// Mitsubishi GX Works2 project: Project1   PLC: FX3G

// global labels: Global1
VAR_GLOBAL
  StartWorkDay AT X007 : BOOL;
  TurnLightAssist AT X011 : BOOL;
  CurrentlyWorking AT Y007 : BOOL;
  yeastInput AT D1100 : REAL;
  yeastInventory AT D1108 : REAL;
  maltInput AT D1102 : REAL;
  maltInventory AT D1110 : REAL;
  hopsInput AT D1104 : REAL;
  hopsInventory AT D1112 : REAL;
  readyBeerPacks AT D1106 : INT;
  startCookingPhase AT X001 : BOOL;
END_VAR
VAR_GLOBAL CONSTANT
  pilsnerMin : INT := 6;
END_VAR
VAR_GLOBAL
  analogInput AT D8280 : INT;
END_VAR
VAR_GLOBAL CONSTANT
  cont400 : INT := 400;
END_VAR
VAR_GLOBAL
  saveAnalog AT D7000 : INT;
  pilsnerCheckAssist AT M0 : BOOL;
  lagerCheckAssist AT M1 : BOOL;
END_VAR
VAR_GLOBAL CONSTANT
  yeastPilsnerMin : REAL := 120;
  maltPilsnerMin : REAL := 6;
  hopsPilsnerMin : REAL := 53;
  cookingTime : INT := 400;
END_VAR
VAR_GLOBAL
  yesPilsnerInventory AT M16 : BOOL;
  CookingTimer AT TC1 : BOOL;
END_VAR
VAR_GLOBAL CONSTANT
  DoneCooking : INT := 40;
END_VAR
VAR_GLOBAL
  Cooking AT TS1 : BOOL;
  CookingProcess AT Y001 : BOOL;
END_VAR
VAR_GLOBAL CONSTANT
  yeastLagerMin : REAL := 150;
  maltLagerMin : REAL := 12;
  hopsLagerMin : REAL := 60;
END_VAR
VAR_GLOBAL
  yesLagerInventory AT M17 : BOOL;
END_VAR
VAR_GLOBAL CONSTANT
  lagerMax : INT := 5;
END_VAR
VAR_GLOBAL
  startFermPhase AT X005 : BOOL;
END_VAR
VAR_GLOBAL CONSTANT
  doneFermPilsner : INT := 40;
END_VAR
VAR_GLOBAL
  FermPilsner AT TC3 : BOOL;
  FermLager AT TC5 : BOOL;
END_VAR
VAR_GLOBAL CONSTANT
  doneFermLager : INT := 30;
END_VAR
VAR_GLOBAL
  FermPilsnerDone AT TS3 : BOOL;
  FermLagerDone AT TS5 : BOOL;
  startBlinking AT M20 : BOOL;
  blinkingHelp AT M21 : BOOL;
  blinkY3 AT TC2 : BOOL;
END_VAR
VAR_GLOBAL CONSTANT
  blinkTime : INT := 5;
END_VAR
VAR_GLOBAL
  blink1 AT TS2 : BOOL;
  lightY3 AT Y003 : BOOL;
  blinkY4 AT TC4 : BOOL;
  blink2 AT TS4 : BOOL;
  lightY4 AT Y004 : BOOL;
  startPackPhase AT X002 : BOOL;
  packBottle AT X000 : BOOL;
  bottlesNum AT CC1 : BOOL;
END_VAR
VAR_GLOBAL CONSTANT
  bottlesPacked : INT := 1;
END_VAR
VAR_GLOBAL
  sixPackNum AT CC2 : BOOL;
END_VAR
VAR_GLOBAL CONSTANT
  sixPacksPacked : INT := 6;
END_VAR
VAR_GLOBAL
  oneBottlePacked AT CS1 : BOOL;
  duringPacking AT Y002 : BOOL;
  doneSixPack AT CS2 : BOOL;
END_VAR
VAR_GLOBAL CONSTANT
  addSixPack : INT := 1;
END_VAR
VAR_GLOBAL
  lackOfProducts AT M19 : BOOL;
  doneSixPacks AT CS2 : BOOL;
  checkYeastForPilsner AT M22 : BOOL;
  checkMaltForPilsner AT M23 : BOOL;
  checkHopsForPilsner AT M24 : BOOL;
  checkYeastForLager AT M25 : BOOL;
  checkMaltForLager AT M26 : BOOL;
  checkHopsForLager AT M27 : BOOL;
  checkYeastForPilsnerEnd AT M70 : BOOL;
  checkMaltForPilsnerEnd AT M71 : BOOL;
  checkHopsForPilsnerEnd AT M72 : BOOL;
  checkYeastForLagerEnd AT M73 : BOOL;
  checkMaltForLagerEnd AT M74 : BOOL;
  checkHopsForLagerEnd AT M75 : BOOL;
  startAnalogOutput AT M100 : BOOL;
END_VAR
VAR_GLOBAL CONSTANT
  constDivide : INT := 40;
END_VAR
VAR_GLOBAL
  analogOutput AT D8282 : INT;
  lackOfProductsEnd AT M50 : BOOL;
END_VAR

// task Task_01 (event TRUE, interval 0, priority 31): POU_01

PROGRAM POU_01
(* structured ladder/FBD written out as ST: instructions are called as NAME(EN, inputs, outputs); _pN, _eN, _tN stand for wires *)
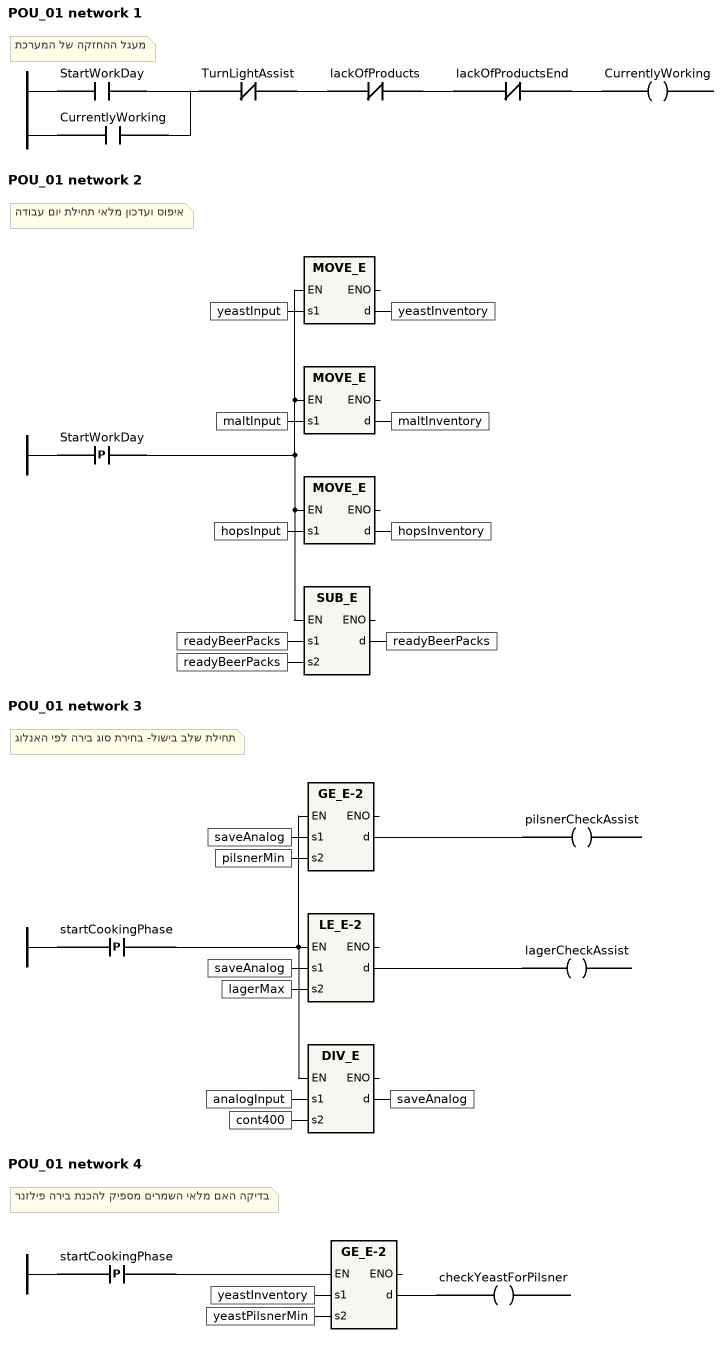
(* network 1 *)
(* מעגל ההחזקה של המערכת *)
CurrentlyWorking := (((StartWorkDay OR CurrentlyWorking) AND NOT TurnLightAssist) AND NOT lackOfProducts) AND NOT lackOfProductsEnd;
(* network 2 *)
(* איפוס ועדכון מלאי תחילת יום עבודה *)
_p1 := LDP(TRUE, StartWorkDay);
MOVE_E(_p1, yeastInput, yeastInventory);
MOVE_E(_p1, maltInput, maltInventory);
MOVE_E(_p1, hopsInput, hopsInventory);
SUB_E(_p1, readyBeerPacks, readyBeerPacks, readyBeerPacks);
(* network 3 *)
(* תחילת שלב בישול- בחירת סוג בירה לפי האנלוג *)
_p1 := LDP(TRUE, startCookingPhase);
DIV_E(_p1, analogInput, cont400, saveAnalog);
GE_E(_p1, saveAnalog, pilsnerMin, _t2);
pilsnerCheckAssist := _t2;
LE_E(_p1, saveAnalog, lagerMax, _t3);
lagerCheckAssist := _t3;
(* network 4 *)
(* בדיקה האם מלאי השמרים מספיק להכנת בירה פילזנר *)
GE_E(LDP(TRUE, startCookingPhase), yeastInventory, yeastPilsnerMin, _t1);
checkYeastForPilsner := _t1;
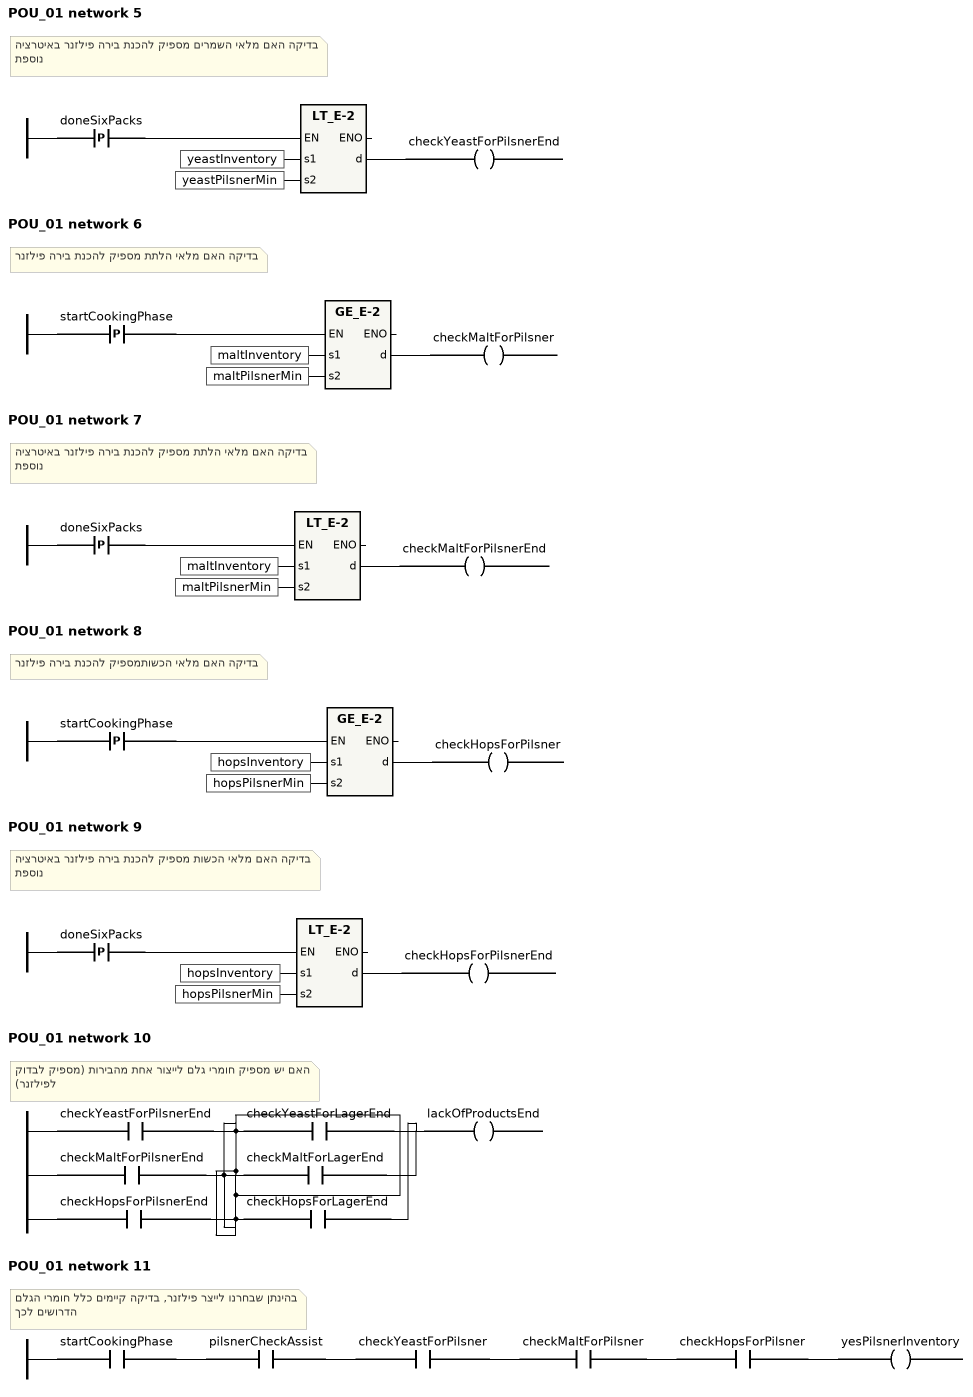
(* network 5 *)
(* בדיקה האם מלאי השמרים מספיק להכנת בירה פילזנר באיטרציה נוספת *)
LT_E(LDP(TRUE, doneSixPacks), yeastInventory, yeastPilsnerMin, _t1);
checkYeastForPilsnerEnd := _t1;
(* network 6 *)
(* בדיקה האם מלאי הלתת מספיק להכנת בירה פילזנר *)
GE_E(LDP(TRUE, startCookingPhase), maltInventory, maltPilsnerMin, _t1);
checkMaltForPilsner := _t1;
(* network 7 *)
(* בדיקה האם מלאי הלתת מספיק להכנת בירה פילזנר באיטרציה נוספת *)
LT_E(LDP(TRUE, doneSixPacks), maltInventory, maltPilsnerMin, _t1);
checkMaltForPilsnerEnd := _t1;
(* network 8 *)
(* בדיקה האם מלאי הכשותמספיק להכנת בירה פילזנר *)
GE_E(LDP(TRUE, startCookingPhase), hopsInventory, hopsPilsnerMin, _t1);
checkHopsForPilsner := _t1;
(* network 9 *)
(* בדיקה האם מלאי הכשות מספיק להכנת בירה פילזנר באיטרציה נוספת *)
LT_E(LDP(TRUE, doneSixPacks), hopsInventory, hopsPilsnerMin, _t1);
checkHopsForPilsnerEnd := _t1;
(* network 10 *)
(* האם יש מספיק חומרי גלם לייצור אחת מהבירות (מספיק לבדוק לפילזנר) *)
_p1 := checkYeastForPilsnerEnd OR checkMaltForPilsnerEnd OR checkHopsForPilsnerEnd;
lackOfProductsEnd := (_p1 AND checkYeastForLagerEnd) OR (_p1 AND checkMaltForLagerEnd) OR (_p1 AND checkHopsForLagerEnd);
(* network 11 *)
(* בהינתן שבחרנו לייצר פילזנר, בדיקה קיימים כלל חומרי הגלם הדרושים לכך *)
yesPilsnerInventory := startCookingPhase AND pilsnerCheckAssist AND checkYeastForPilsner AND checkMaltForPilsner AND checkHopsForPilsner;
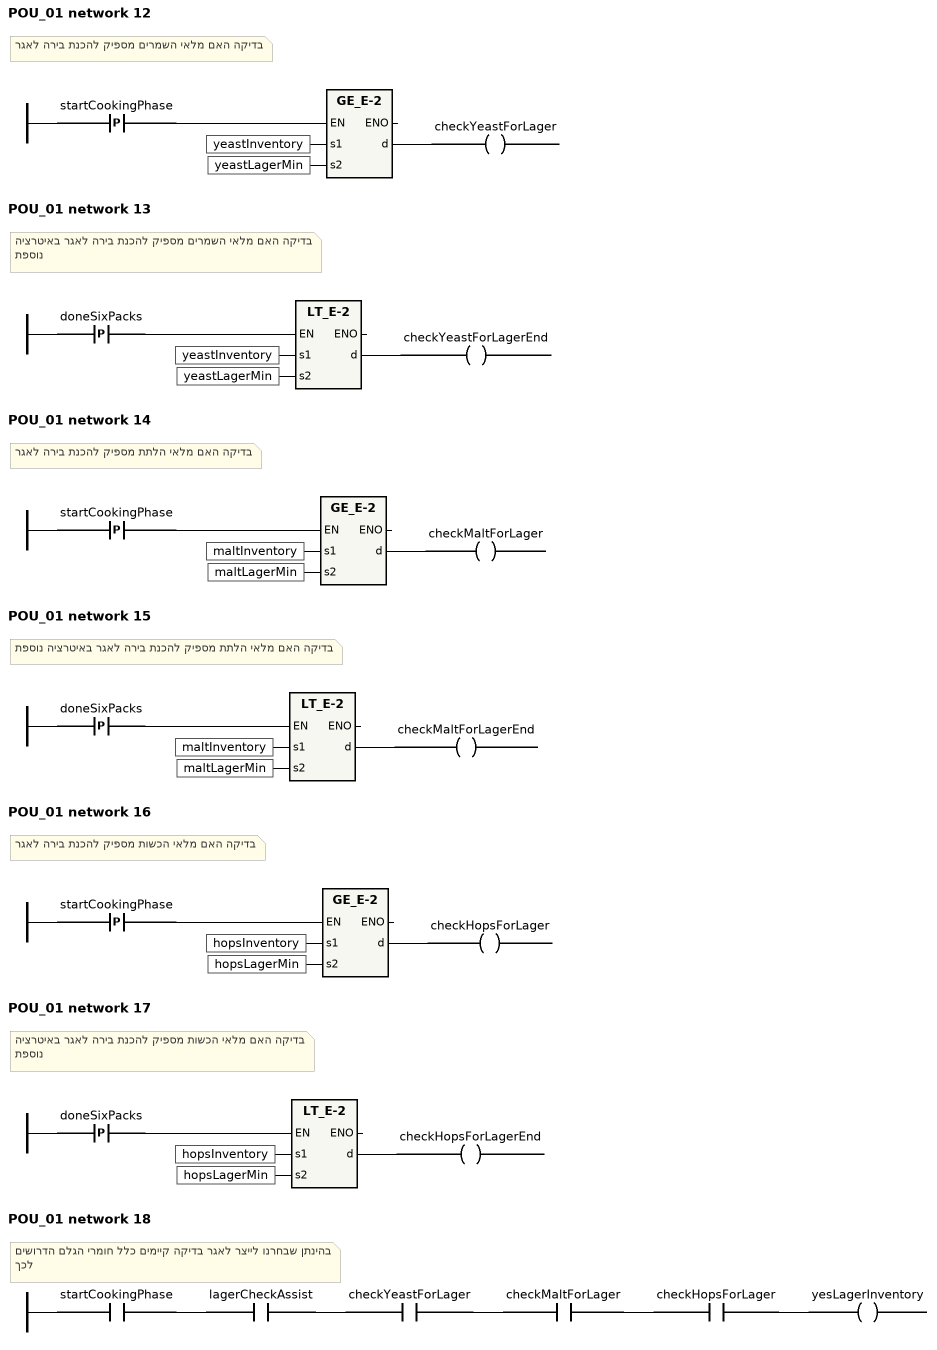
(* network 12 *)
(* בדיקה האם מלאי השמרים מספיק להכנת בירה לאגר *)
GE_E(LDP(TRUE, startCookingPhase), yeastInventory, yeastLagerMin, _t1);
checkYeastForLager := _t1;
(* network 13 *)
(* בדיקה האם מלאי השמרים מספיק להכנת בירה לאגר באיטרציה נוספת *)
LT_E(LDP(TRUE, doneSixPacks), yeastInventory, yeastLagerMin, _t1);
checkYeastForLagerEnd := _t1;
(* network 14 *)
(* בדיקה האם מלאי הלתת מספיק להכנת בירה לאגר *)
GE_E(LDP(TRUE, startCookingPhase), maltInventory, maltLagerMin, _t1);
checkMaltForLager := _t1;
(* network 15 *)
(* בדיקה האם מלאי הלתת מספיק להכנת בירה לאגר באיטרציה נוספת *)
LT_E(LDP(TRUE, doneSixPacks), maltInventory, maltLagerMin, _t1);
checkMaltForLagerEnd := _t1;
(* network 16 *)
(* בדיקה האם מלאי הכשות מספיק להכנת בירה לאגר *)
GE_E(LDP(TRUE, startCookingPhase), hopsInventory, hopsLagerMin, _t1);
checkHopsForLager := _t1;
(* network 17 *)
(* בדיקה האם מלאי הכשות מספיק להכנת בירה לאגר באיטרציה נוספת *)
LT_E(LDP(TRUE, doneSixPacks), hopsInventory, hopsLagerMin, _t1);
checkHopsForLagerEnd := _t1;
(* network 18 *)
(* בהינתן שבחרנו לייצר לאגר בדיקה קיימים כלל חומרי הגלם הדרושים לכך *)
yesLagerInventory := startCookingPhase AND lagerCheckAssist AND checkYeastForLager AND checkMaltForLager AND checkHopsForLager;
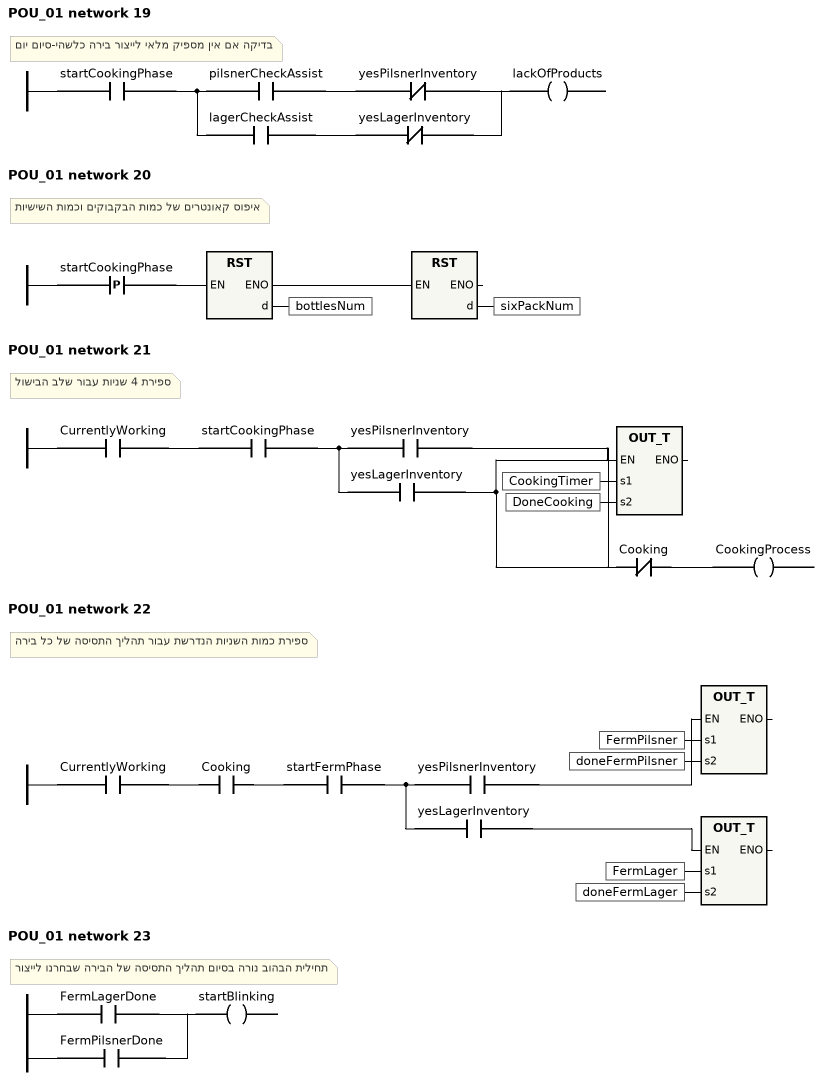
(* network 19 *)
(* בדיקה אם אין מספיק מלאי לייצור בירה כלשהי-סיום יום *)
lackOfProducts := (startCookingPhase AND pilsnerCheckAssist AND NOT yesPilsnerInventory) OR (startCookingPhase AND lagerCheckAssist AND NOT yesLagerInventory);
(* network 20 *)
(* איפוס קאונטרים של כמות הבקבוקים וכמות השישיות *)
_e1 := RST(LDP(TRUE, startCookingPhase), bottlesNum);
RST(_e1, sixPackNum);
(* network 21 *)
(* ספירת 4 שניות עבור שלב הבישול *)
_p1 := CurrentlyWorking AND startCookingPhase;
_p2 := (_p1 AND yesPilsnerInventory) OR (_p1 AND yesLagerInventory);
CookingProcess := _p2 AND NOT Cooking;
OUT_T(_p2, CookingTimer, DoneCooking);
(* network 22 *)
(* ספירת כמות השניות הנדרשת עבור תהליך התסיסה של כל בירה *)
_p1 := CurrentlyWorking AND Cooking AND startFermPhase;
OUT_T(_p1 AND yesPilsnerInventory, FermPilsner, doneFermPilsner);
OUT_T(_p1 AND yesLagerInventory, FermLager, doneFermLager);
(* network 23 *)
(* תחילית הבהוב נורה בסיום תהליך התסיסה של הבירה שבחרנו לייצור *)
startBlinking := FermLagerDone OR FermPilsnerDone;
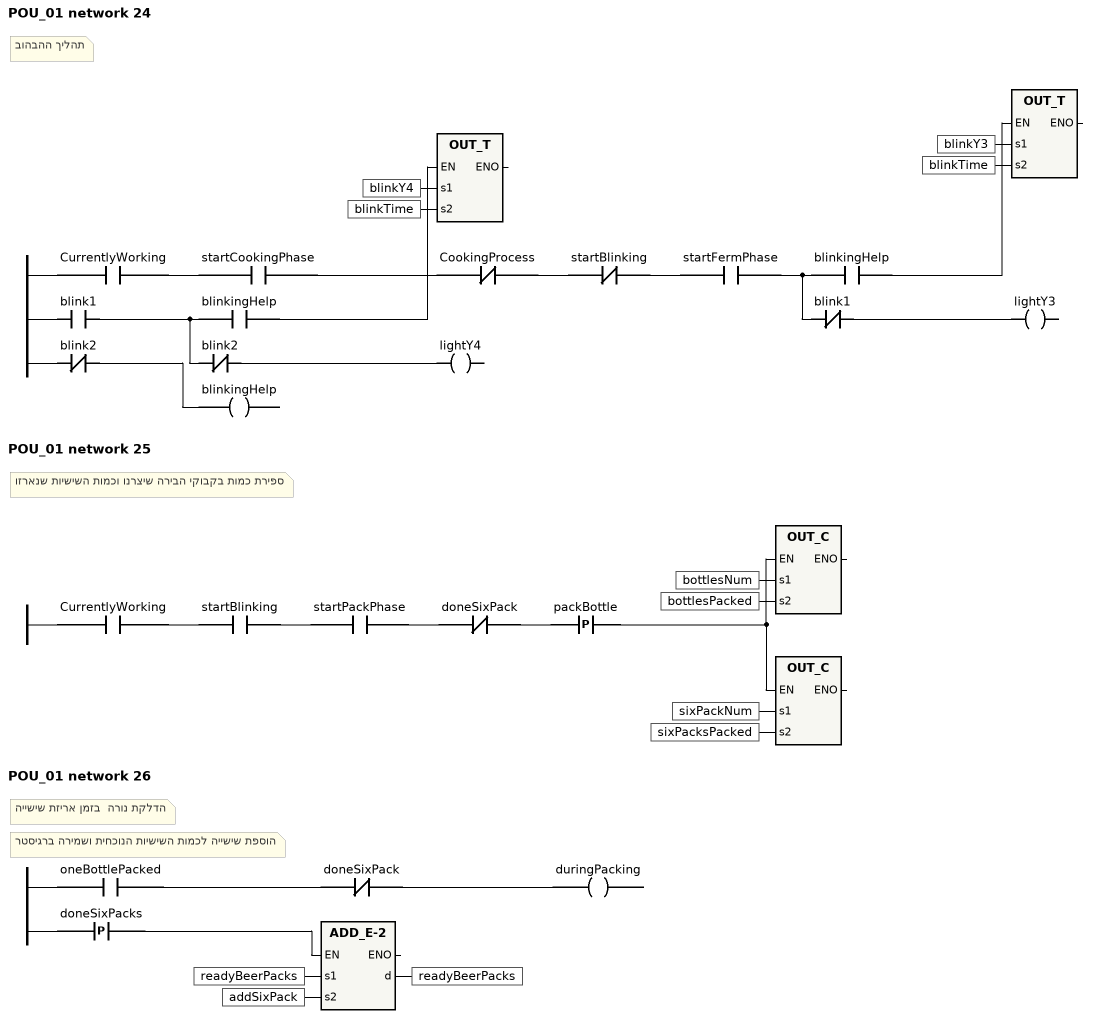
(* network 24 *)
(* תהליך ההבהוב *)
_p1 := CurrentlyWorking AND startCookingPhase AND NOT CookingProcess AND NOT startBlinking AND startFermPhase;
OUT_T(_p1 AND blinkingHelp, blinkY3, blinkTime);
lightY3 := _p1 AND NOT blink1;
OUT_T(blink1 AND blinkingHelp, blinkY4, blinkTime);
lightY4 := blink1 AND NOT blink2;
blinkingHelp := NOT blink2;
(* network 25 *)
(* ספירת כמות בקבוקי הבירה שיצרנו וכמות השישיות שנארזו *)
_p1 := CurrentlyWorking AND startBlinking AND startPackPhase AND NOT doneSixPack AND LDP(TRUE, packBottle);
OUT_C(_p1, bottlesNum, bottlesPacked);
OUT_C(_p1, sixPackNum, sixPacksPacked);
(* network 26 *)
(* הדלקת נורה  בזמן אריזת שישייה *)
(* הוספת שישייה לכמות השישיות הנוכחית ושמירה ברגיסטר *)
duringPacking := oneBottlePacked AND NOT doneSixPack;
ADD_E(LDP(TRUE, doneSixPacks), readyBeerPacks, addSixPack, readyBeerPacks);
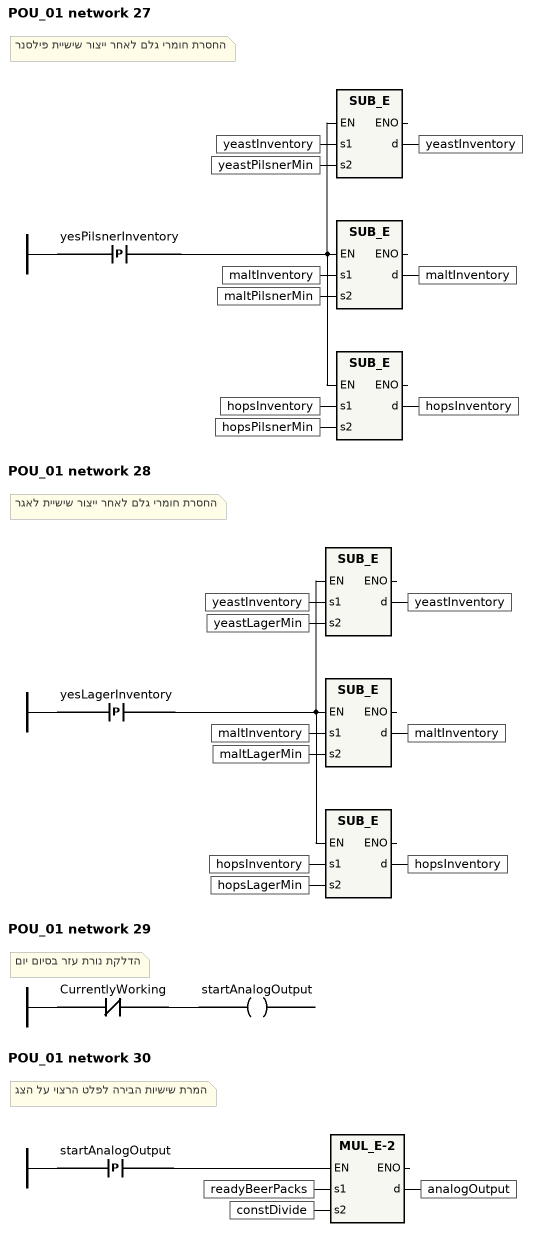
(* network 27 *)
(* החסרת חומרי גלם לאחר ייצור שישיית פילסנר *)
_p1 := LDP(TRUE, yesPilsnerInventory);
SUB_E(_p1, yeastInventory, yeastPilsnerMin, yeastInventory);
SUB_E(_p1, maltInventory, maltPilsnerMin, maltInventory);
SUB_E(_p1, hopsInventory, hopsPilsnerMin, hopsInventory);
(* network 28 *)
(* החסרת חומרי גלם לאחר ייצור שישיית לאגר *)
_p1 := LDP(TRUE, yesLagerInventory);
SUB_E(_p1, yeastInventory, yeastLagerMin, yeastInventory);
SUB_E(_p1, maltInventory, maltLagerMin, maltInventory);
SUB_E(_p1, hopsInventory, hopsLagerMin, hopsInventory);
(* network 29 *)
(* הדלקת נורת עזר בסיום יום *)
startAnalogOutput := NOT CurrentlyWorking;
(* network 30 *)
(* המרת שישיות הבירה לפלט הרצוי על הצג *)
MUL_E(LDP(TRUE, startAnalogOutput), readyBeerPacks, constDivide, analogOutput);
END_PROGRAM
